(* Logix 5000 project; controller cal1615 1756-L62 rev 20.11; software revision 20.05; part 41 of 82 *)
(* tags used below, declared in another part *)
   FAULT : BOOL;   // Fault AFI
   p01_recipe_active : recipe;   // Active Recipe
   p01r02_plc_scan_time_in_sec : REAL;   // System PLC Scan Time in Seconds
   p01r09 : routine;   // System Modes
   p01r09_pb_global_reset : BOOL;   // System Modes PB: Global Fault Reset
   p01r12_master_ramped_speed : REAL;   // System Line Accel Decel Control Master Ramped Speed
   p01r13_line_running : BOOL;   // System Line Start Sequence Line Running
   p01r13_line_slow_ramp : BOOL;   // System Line Start Sequence Start Line to Slow Speed
   p01r13_permissive_drives : BOOL;   // System Line Start Sequence Permissive Drives
   p02_dint_from_hmi : hmi_dint;
   p20_acc_fill_prs : REAL;   // Upper Poly Letoff Modes A Toggle
   p20_acc_tens_prs : REAL;   // Letoff Accumulator Pressure Tension Setpoint
   p20_ai_lc01 : REAL;   // Letoff Analog Input Line Tension Load Cell Splicer
   p20_ai_loa_speed : REAL;   // Letoff Inputs Letoff A VFD Surface Speed
   p20_ao_acc_ctr_prs : REAL;   // Letoff Analog Output Accumulator Counter Pressure
   p20_ao_acc_ten_prs : REAL;   // Letoff Analog Output Accumulator Tension Pressure
   p20_ao_loa_selected_speed : REAL;   // Letoff Output Selected Speed
   p20_ao_loa_torque : REAL;
   p20_di_acc_empty : BOOL;   // Letoff Digital Input Letoff Accumulator Empty Position
   p20_di_acc_full : BOOL;   // Letoff Digital Input Letoff Accumulator Full Control Position
   p20_di_loa_active : BOOL;   // Letoff Digital Input Letoff A Active
   p20_di_loa_fwd_dir : BOOL;   // Letoff Digital Inputs PB: Letoff A Jog FWD
   p20_di_loa_jog : BOOL;   // Letoff Digital Inputs PB: Letoff A Jog REV
   p20_di_loa_start : BOOL;   // Letoff Digital Input PB: Letoff A Start
   p20_di_loa_stop : BOOL;   // Letoff Digital Input PB: Letoff A Stop Stop = 0
   p20_di_lof_acc_fill : BOOL;   // Letoff Digital Input PB: Accumulator Fill
   p20_do_acc_enable_tension : BOOL;   // Letoff Digital Output Enable Accumulator Lift Tension
   p20_do_close_nip : BOOL;   // Letoff Digital Output Feedroll Roll Nip Close
   p20_param_acc_auto_fill : REAL;
   p20_param_acc_ctr_prs : REAL;   // Letoff Parameter Carriage Counter Pressure Setpoint
   p20_param_acc_empty_prs : REAL;
   p20_param_acc_fast_accel : REAL;
   p20_param_acc_fast_decel : REAL;
   p20_param_acc_fill_ctr_prs : REAL;
   p20_param_acc_high_prs : REAL;   // Letoff Parameter High Pressure Setpoint
   p20_param_acc_init_high_prs : REAL;
   p20_param_acc_init_low_prs : REAL;
   p20_param_acc_init_prs : REAL;   // Letoff Accumulator Initial Pressure for Ramp
   p20_param_acc_med_accel : REAL;
   p20_param_acc_med_decel : REAL;
   p20_param_acc_pid_accel : REAL;
   p20_param_acc_pid_decel : REAL;
   p20_param_acc_pos_prs : REAL;
   p20_param_acc_slow_accel : REAL;
   p20_param_acc_slow_decel : REAL;
   p20_param_empty_pct : REAL;
   p20_param_high_accel_rate : REAL;
   p20_param_high_ctrl_pct : REAL;   // Letoff Parameter High Accumulator Control Position
   p20_param_high_decel_rate : REAL;
   p20_param_high_low_ctrl_pct : REAL;   // Letoff Accumulator High Control Position Low Limit
   p20_param_jog_accel_rate : REAL;
   p20_param_jog_decel_rate : REAL;
   p20_param_letoff_jog_speed : REAL;
   p20_param_lof_fast_fill : REAL;
   p20_param_lof_slow_fill : REAL;
   p20_param_lof_stop_fill : REAL;
   p20_param_low_ctrl_pct : REAL;   // Letoff Parameter Low Accumulator Control Position
   p20_param_low_low_ctrl_pct : REAL;
   p20_param_norm_accel_rate : REAL;
   p20_param_norm_decel_rate : REAL;   // Letoff Parameter Letoff A Decel Rate
   p20_param_prs_accel_rate : REAL;   // Letoff Accumulator Accel/Decel Ramp Accel Rate
   p20_param_prs_decel_rate : REAL;   // Letoff Accumulator Accel/Decel Ramp Decel Rate
   p20_param_run_torque : REAL;
   p20_vfd_di_loa : acs800_di_normal;   // Letoff A VFD Inputs
   p20_vfd_do_loa : acs800_do_normal;   // Letoff A VFD Outputs
   p20_zero_tension_prs : REAL;
   p20r01 : routine;   // Letoff Main
   p20r09_accumulator_auto : BOOL;   // Letoff Modes Accumulator Auto Mode
   p20r10_pid_psn : PID;   // Letoff Letoff Position Control PID
   p20r10_speed_offset : REAL;   // Letoff Letoff Speed Control Speed Offset
   p20r11_request_close_nip : BOOL;   // Letoff Feedroll Request Close Feedroll Nip Roll
   p20r13 : routine;   // Letoff Accum Control
   p20r13_acc_top_pos : REAL;   // Upper Poly Letoff Modes Letoff B Tension Mode
   p20r13_ai_acc_pct : REAL;   // Letoff Accumulator Pct Full
   p20r13_enc : SYS_ENC;   // Letoff Accumulator Encoder
   p20r13_ramp_tension_pressure : SYS_ACC_DEC_RAMP;   // Letoff Accumulator Tension Pressure Ramp
   p20r13_request_fill : BOOL;   // Letoff Accumulator Request Fill
   p20r13_selected_pressure : REAL;   // Letoff Accumulator Selected Pressure
   p20r13_state : DINT;   // Letoff Accumulator State
   p20r13_status : DINT;   // Letoff Accumulator Fill Status
   p20r13_timer_fault : TIMER[4];   // Letoff Accum Control Fault Delay
   p20r13_timer_warning : TIMER[4];   // Letoff Accum Control Warning Delay
   p20r14_acc_request_tension_ctrl : BOOL;   // Letoff Accumulator Fill Pressure Request Tension Control
   p20r15 : routine;   // Letoff Letoff A VFD
   p20r15_loa_accel : REAL;   // Letoff Letoff A VFD Accel Rate ORG: 100
   p20r15_loa_accel_decel_ramp : SYS_ACC_DEC_RAMP;   // Letoff Letoff A VFD Accel Decel Ramp
   p20r15_loa_decel : REAL;   // Letoff Letoff A VFD Decel Rate ORG: 20
   p20r15_loa_on : BOOL;   // Letoff Letoff A VFD On
   p20r15_loa_selected_speed : REAL;   // Letoff Letoff A VFD Selected Speed
   p20r15_permissive_run : BOOL;   // Letoff Letoff A VFD Permissive Run
   p20r15_request_jog_fwd : BOOL;   // Letoff Letoff A VFD Request Jog FWD
   p20r15_request_jog_rev : BOOL;   // Letoff Letoff A VFD Request Jog REV
   p20r15_request_over_speed : BOOL;   // Letoff Letoff A VFD Request Accumulator Over-Speed
   p20r15_request_position : BOOL;   // Letoff Letoff A VFD Request Accumulator Position Control
   p20r15_request_stop : BOOL;   // Letoff Letoff A VFD Request Stop
   p20r15_request_tension : BOOL;   // Letoff Letoff A VFD Request Tension
   p20r15_request_thread_fwd : BOOL;
   p20r15_request_thread_rev : BOOL;
   p20r15_timer_fault : TIMER[10];   // Letoff Letoff A VFD Fault Timer
   p20r15_zero_speed : BOOL;   // Letoff Letoff A VFD At Zero Speed
   p20r17_letoff_avg_diam_inch : REAL;   // Letoff Letoff Diameter Calc Average Diameter [in]
   p22_ao_selected_speed : REAL;   // Tension Stand 1 VFD Selected Speed
   p22r11_request_thread_fwd : BOOL;   // Tension Stand 1 VFD Request Thread FWD
   p22r11_request_thread_rev : BOOL;   // Tension Stand 1 VFD Request Thread REV
   p25r11_request_thread_fwd : BOOL;   // Tension Stand 2 VFD Request Thread FWD
   p25r11_request_thread_rev : BOOL;   // Tension Stand 2 VFD Request Thread REV
   p27r01 : routine;   // Winder Main
(* P20_Letoff, continued *)

ROUTINE R13_Accumulator   (* ladder *)
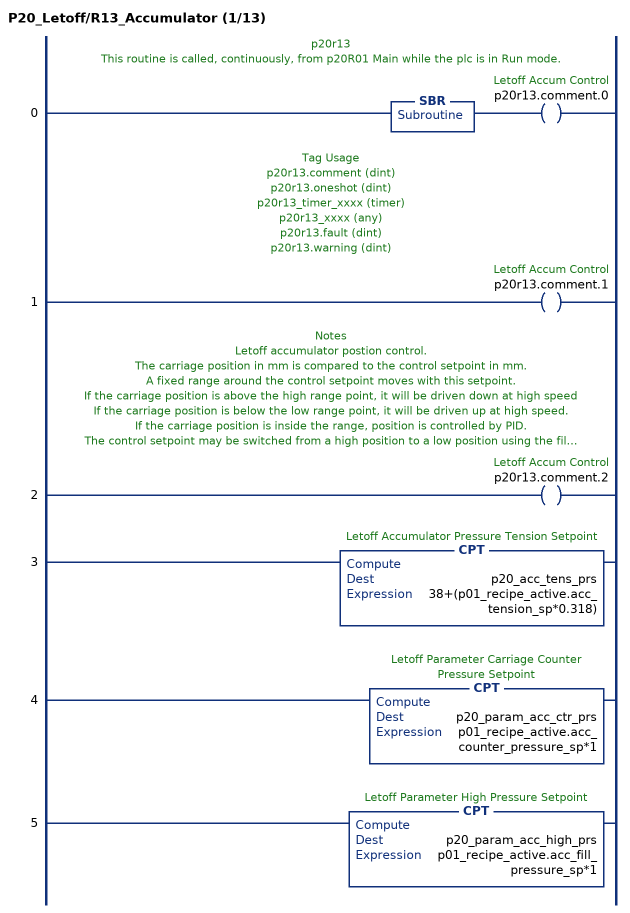
   // p20r13
   // This routine is called, continuously, from p20R01 Main while the plc is in Run mode.
   0: SBR()OTE(p20r13.comment.0);
   // Tag Usage
   // p20r13.comment (dint)
   // p20r13.oneshot (dint)
   // p20r13_timer_xxxx (timer)
   // p20r13_xxxx (any)
   // p20r13.fault (dint)
   // p20r13.warning (dint)
   1: OTE(p20r13.comment.1);
   // Notes
   // Letoff accumulator postion control.
   // The carriage position in mm is compared to the control setpoint in mm.
   // A fixed range around the control setpoint moves with this setpoint.
   // If the carriage position is above the high range point, it will be driven down at high speed
   // If the carriage position is below the low range point, it will be driven up at high speed.
   // If the carriage position is inside the range, position is controlled by PID.
   // The control setpoint may be switched from a high position to a low position using the fill accumulator function.
   2: OTE(p20r13.comment.2);
   3: CPT(p20_acc_tens_prs,38+(p01_recipe_active.acc_tension_sp*0.318));
   4: CPT(p20_param_acc_ctr_prs,p01_recipe_active.acc_counter_pressure_sp*1);
   5: CPT(p20_param_acc_high_prs,p01_recipe_active.acc_fill_pressure_sp*1);
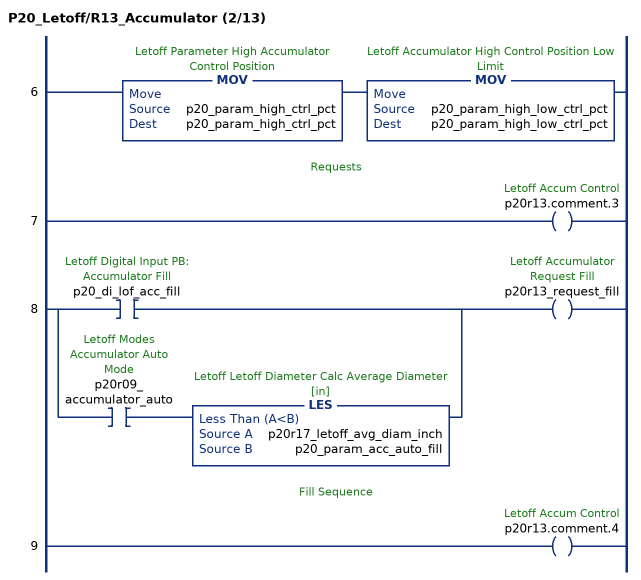
   6: MOV(p20_param_high_ctrl_pct,p20_param_high_ctrl_pct)MOV(p20_param_high_low_ctrl_pct,p20_param_high_low_ctrl_pct);
   // Requests
   7: OTE(p20r13.comment.3);
   8: [XIC(p20_di_lof_acc_fill) ,XIC(p20r09_accumulator_auto) LES(p20r17_letoff_avg_diam_inch,p20_param_acc_auto_fill) ]OTE(p20r13_request_fill);
   // Fill Sequence
   9: OTE(p20r13.comment.4);
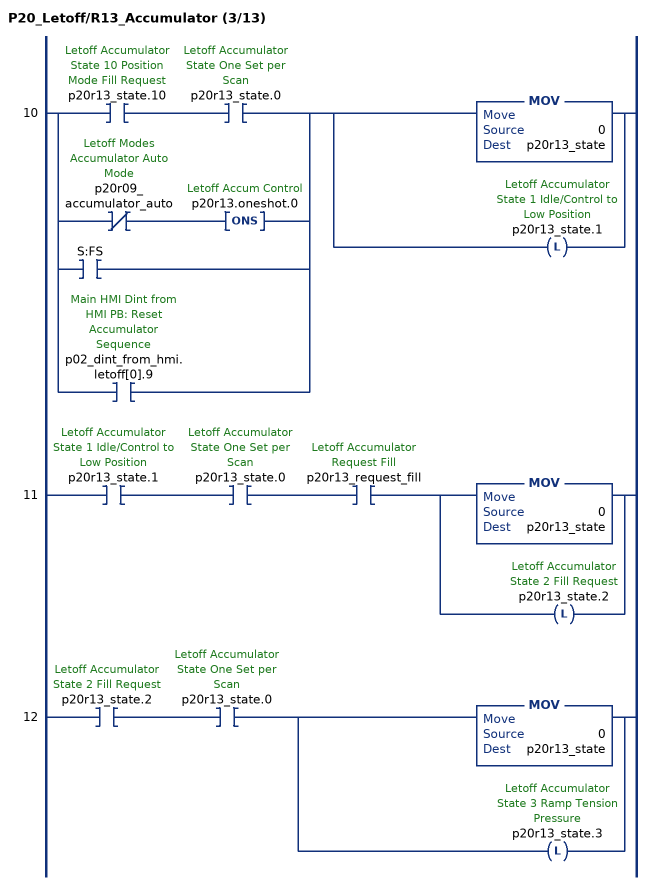
   10: [XIC(p20r13_state.10) XIC(p20r13_state.0) ,XIO(p20r09_accumulator_auto) ONS(p20r13.oneshot.0) ,XIC(S:FS) ,XIC(p02_dint_from_hmi.letoff[0].9) ][MOV(0,p20r13_state) ,OTL(p20r13_state.1) ];
   11: XIC(p20r13_state.1)XIC(p20r13_state.0)XIC(p20r13_request_fill)[MOV(0,p20r13_state) ,OTL(p20r13_state.2) ];
   12: XIC(p20r13_state.2)XIC(p20r13_state.0)[MOV(0,p20r13_state) ,OTL(p20r13_state.3) ];
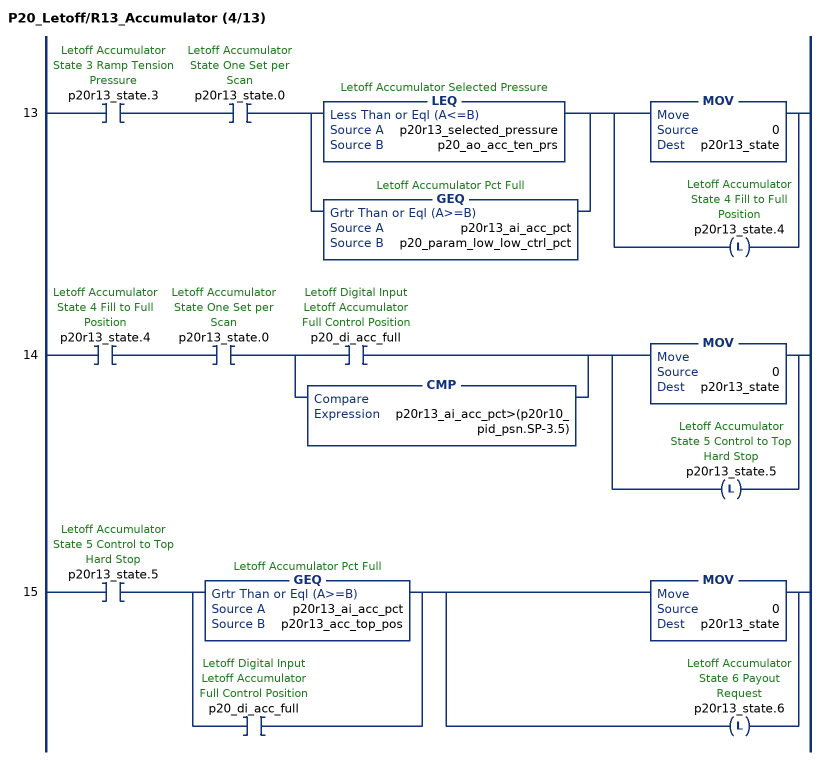
   13: XIC(p20r13_state.3)XIC(p20r13_state.0)[LEQ(p20r13_selected_pressure,p20_ao_acc_ten_prs) ,GEQ(p20r13_ai_acc_pct,p20_param_low_low_ctrl_pct) ][MOV(0,p20r13_state) ,OTL(p20r13_state.4) ];
   14: XIC(p20r13_state.4)XIC(p20r13_state.0)[XIC(p20_di_acc_full) ,CMP(p20r13_ai_acc_pct>(p20r10_pid_psn.SP-3.5)) ][MOV(0,p20r13_state) ,OTL(p20r13_state.5) ];
   15: XIC(p20r13_state.5)[GEQ(p20r13_ai_acc_pct,p20r13_acc_top_pos) ,XIC(p20_di_acc_full) ][MOV(0,p20r13_state) ,OTL(p20r13_state.6) ];
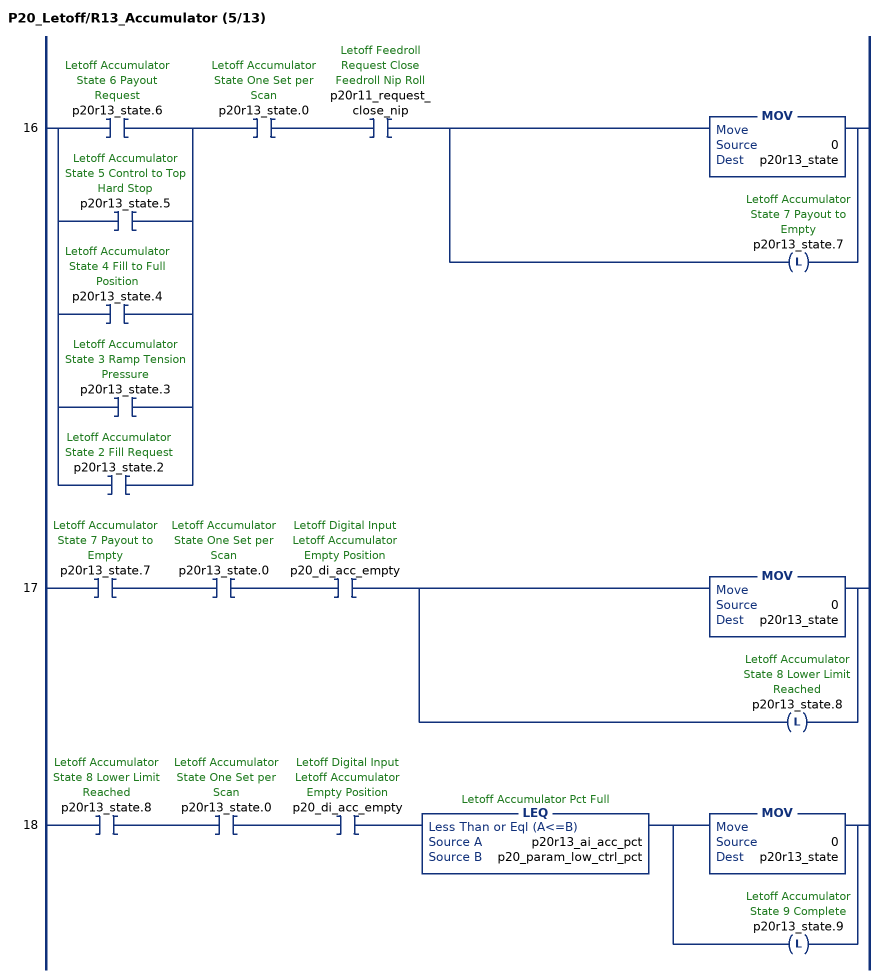
   16: [XIC(p20r13_state.6) ,XIC(p20r13_state.5) ,XIC(p20r13_state.4) ,XIC(p20r13_state.3) ,XIC(p20r13_state.2) ]XIC(p20r13_state.0)XIC(p20r11_request_close_nip)[MOV(0,p20r13_state) ,OTL(p20r13_state.7) ];
   17: XIC(p20r13_state.7)XIC(p20r13_state.0)XIC(p20_di_acc_empty)[MOV(0,p20r13_state) ,OTL(p20r13_state.8) ];
   18: XIC(p20r13_state.8)XIC(p20r13_state.0)XIC(p20_di_acc_empty)LEQ(p20r13_ai_acc_pct,p20_param_low_ctrl_pct)[MOV(0,p20r13_state) ,OTL(p20r13_state.9) ];
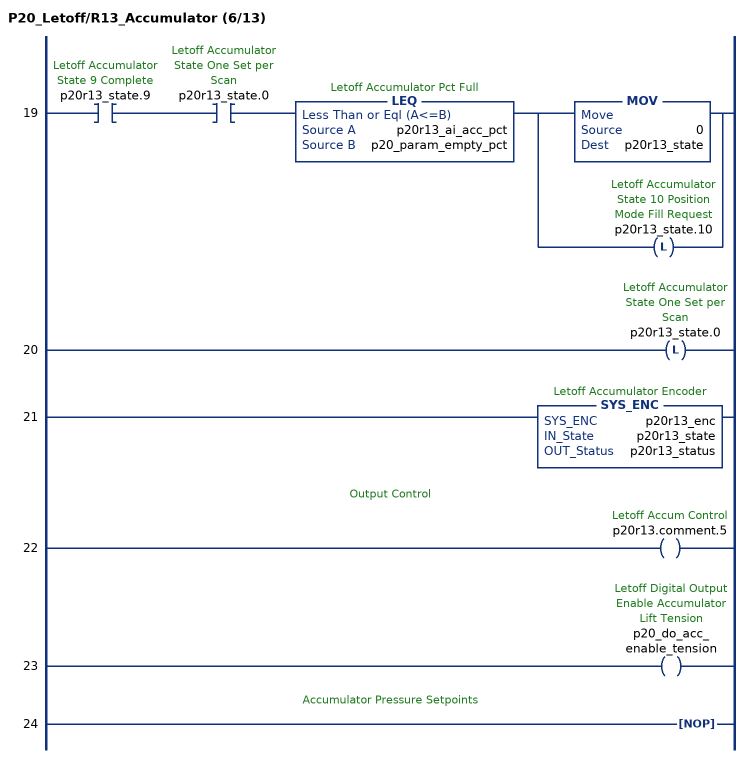
   19: XIC(p20r13_state.9)XIC(p20r13_state.0)LEQ(p20r13_ai_acc_pct,p20_param_empty_pct)[MOV(0,p20r13_state) ,OTL(p20r13_state.10) ];
   20: OTL(p20r13_state.0);
   21: SYS_ENC(p20r13_enc,p20r13_state,p20r13_status);
   // Output Control
   22: OTE(p20r13.comment.5);
   23: OTE(p20_do_acc_enable_tension);
   // Accumulator Pressure Setpoints
   24: NOP();
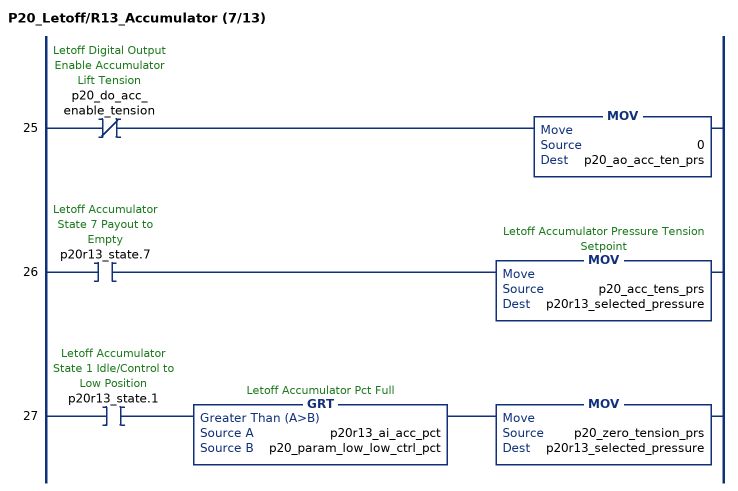
   25: XIO(p20_do_acc_enable_tension)MOV(0,p20_ao_acc_ten_prs);
   26: XIC(p20r13_state.7)MOV(p20_acc_tens_prs,p20r13_selected_pressure);
   27: XIC(p20r13_state.1)GRT(p20r13_ai_acc_pct,p20_param_low_low_ctrl_pct)MOV(p20_zero_tension_prs,p20r13_selected_pressure);
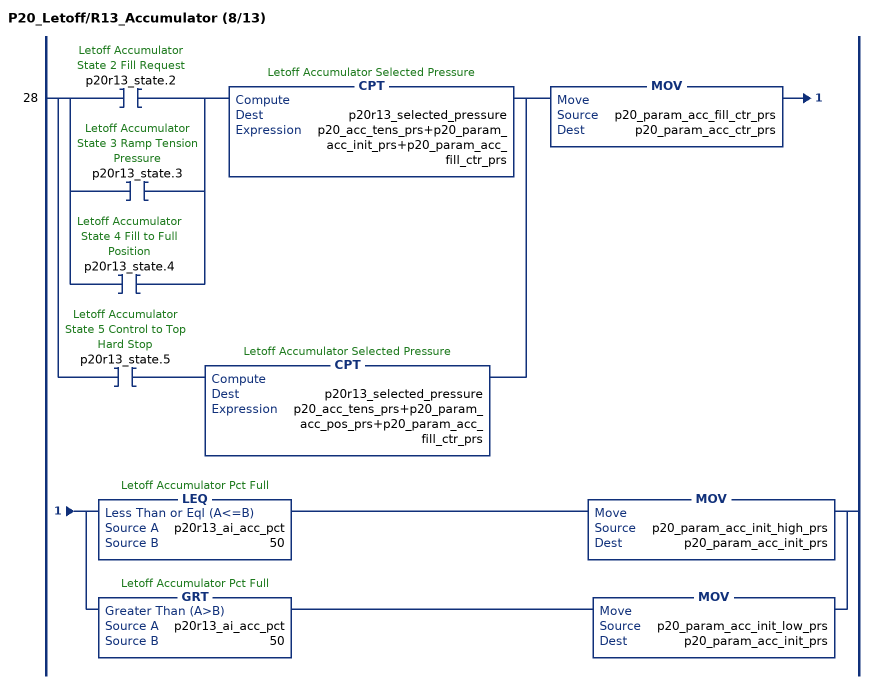
   28: [[XIC(p20r13_state.2) ,XIC(p20r13_state.3) ,XIC(p20r13_state.4) ] CPT(p20r13_selected_pressure,p20_acc_tens_prs+p20_param_acc_init_prs+p20_param_acc_fill_ctr_prs) ,XIC(p20r13_state.5) CPT(p20r13_selected_pressure,p20_acc_tens_prs+p20_param_acc_pos_prs+p20_param_acc_fill_ctr_prs) ]MOV(p20_param_acc_fill_ctr_prs,p20_param_acc_ctr_prs)[LEQ(p20r13_ai_acc_pct,50) MOV(p20_param_acc_init_high_prs,p20_param_acc_init_prs) ,GRT(p20r13_ai_acc_pct,50) MOV(p20_param_acc_init_low_prs,p20_param_acc_init_prs) ];
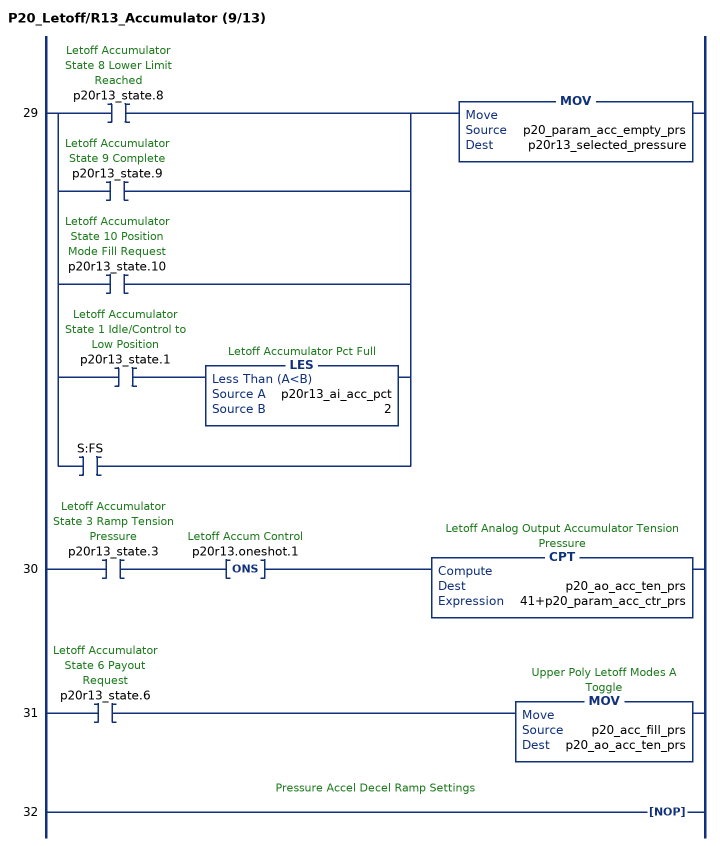
   29: [XIC(p20r13_state.8) ,XIC(p20r13_state.9) ,XIC(p20r13_state.10) ,XIC(p20r13_state.1) LES(p20r13_ai_acc_pct,2) ,XIC(S:FS) ]MOV(p20_param_acc_empty_prs,p20r13_selected_pressure);
   30: XIC(p20r13_state.3)ONS(p20r13.oneshot.1)CPT(p20_ao_acc_ten_prs,41+p20_param_acc_ctr_prs);
   31: XIC(p20r13_state.6)MOV(p20_acc_fill_prs,p20_ao_acc_ten_prs);
   // Pressure Accel Decel Ramp Settings
   32: NOP();
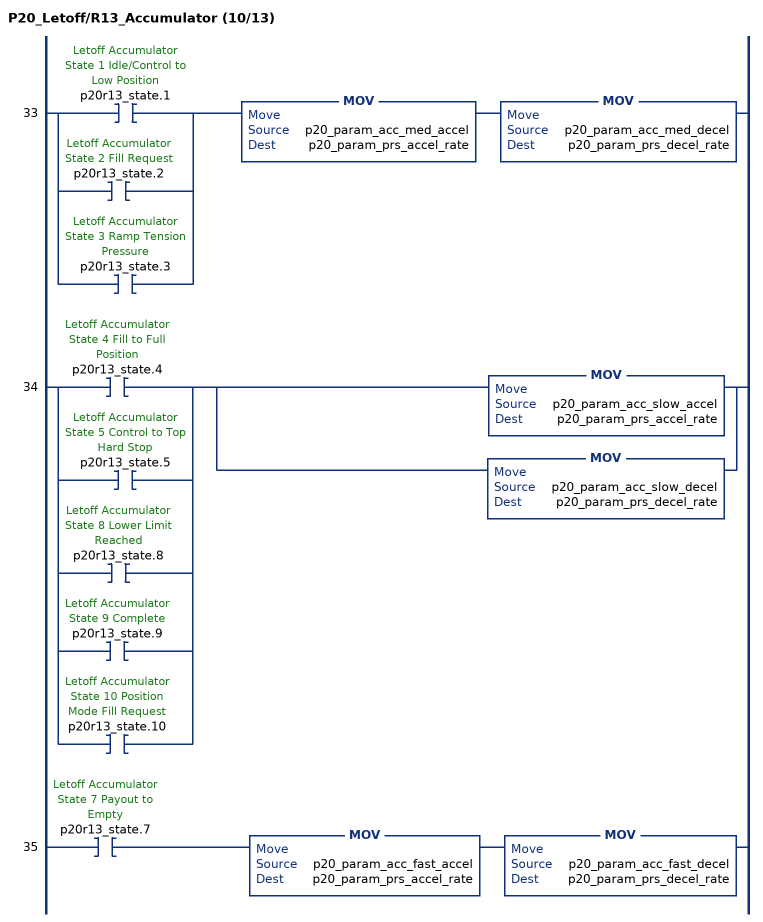
   33: [XIC(p20r13_state.1) ,XIC(p20r13_state.2) ,XIC(p20r13_state.3) ]MOV(p20_param_acc_med_accel,p20_param_prs_accel_rate)MOV(p20_param_acc_med_decel,p20_param_prs_decel_rate);
   34: [XIC(p20r13_state.4) ,XIC(p20r13_state.5) ,XIC(p20r13_state.8) ,XIC(p20r13_state.9) ,XIC(p20r13_state.10) ][MOV(p20_param_acc_slow_accel,p20_param_prs_accel_rate) ,MOV(p20_param_acc_slow_decel,p20_param_prs_decel_rate) ];
   35: XIC(p20r13_state.7)MOV(p20_param_acc_fast_accel,p20_param_prs_accel_rate)MOV(p20_param_acc_fast_decel,p20_param_prs_decel_rate);
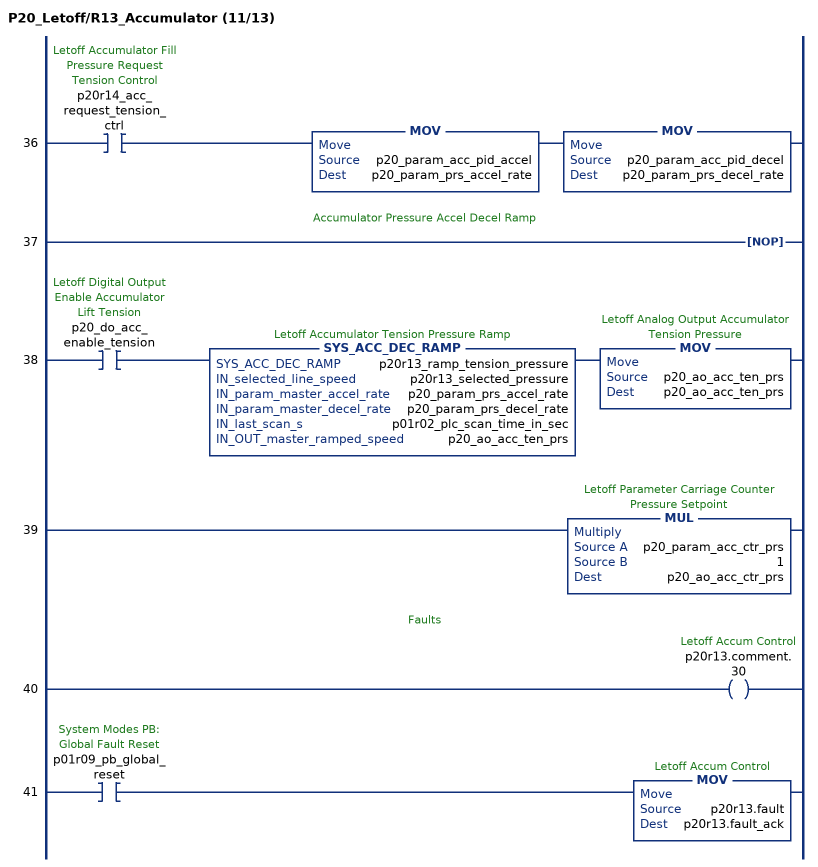
   36: XIC(p20r14_acc_request_tension_ctrl)MOV(p20_param_acc_pid_accel,p20_param_prs_accel_rate)MOV(p20_param_acc_pid_decel,p20_param_prs_decel_rate);
   // Accumulator Pressure Accel Decel Ramp
   37: NOP();
   38: XIC(p20_do_acc_enable_tension)SYS_ACC_DEC_RAMP(p20r13_ramp_tension_pressure,p20r13_selected_pressure,p20_param_prs_accel_rate,p20_param_prs_decel_rate,p01r02_plc_scan_time_in_sec,p20_ao_acc_ten_prs)MOV(p20_ao_acc_ten_prs,p20_ao_acc_ten_prs);
   39: MUL(p20_param_acc_ctr_prs,1,p20_ao_acc_ctr_prs);
   // Faults
   40: OTE(p20r13.comment.30);
   41: XIC(p01r09_pb_global_reset)MOV(p20r13.fault,p20r13.fault_ack);
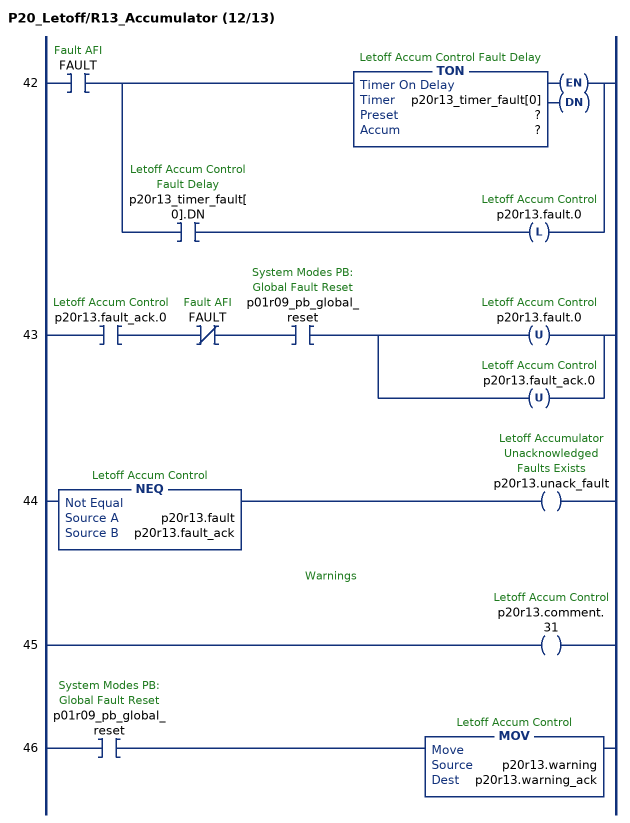
   42: XIC(FAULT)[TON(p20r13_timer_fault[0],?,?) ,XIC(p20r13_timer_fault[0].DN) OTL(p20r13.fault.0) ];
   43: XIC(p20r13.fault_ack.0)XIO(FAULT)XIC(p01r09_pb_global_reset)[OTU(p20r13.fault.0) ,OTU(p20r13.fault_ack.0) ];
   44: NEQ(p20r13.fault,p20r13.fault_ack)OTE(p20r13.unack_fault);
   // Warnings
   45: OTE(p20r13.comment.31);
   46: XIC(p01r09_pb_global_reset)MOV(p20r13.warning,p20r13.warning_ack);
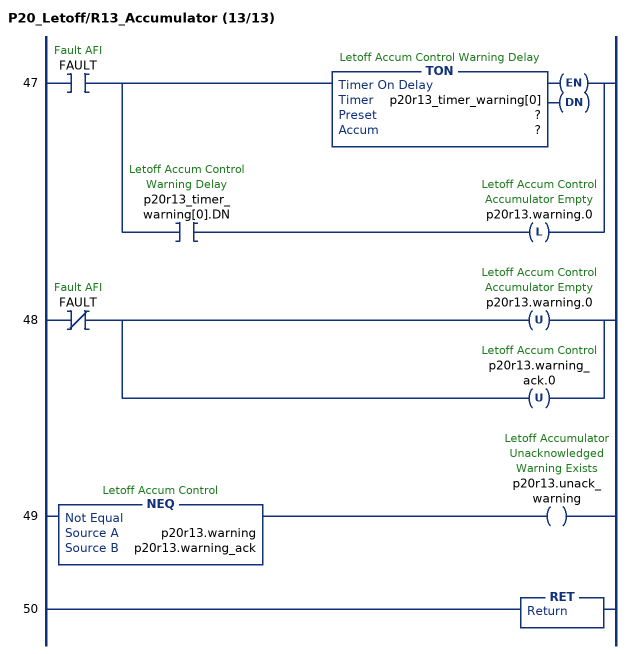
   47: XIC(FAULT)[TON(p20r13_timer_warning[0],?,?) ,XIC(p20r13_timer_warning[0].DN) OTL(p20r13.warning.0) ];
   48: XIO(FAULT)[OTU(p20r13.warning.0) ,OTU(p20r13.warning_ack.0) ];
   49: NEQ(p20r13.warning,p20r13.warning_ack)OTE(p20r13.unack_warning);
   50: RET();
END_ROUTINE

ROUTINE R15_Letoff_A_VFD   (* ladder *)
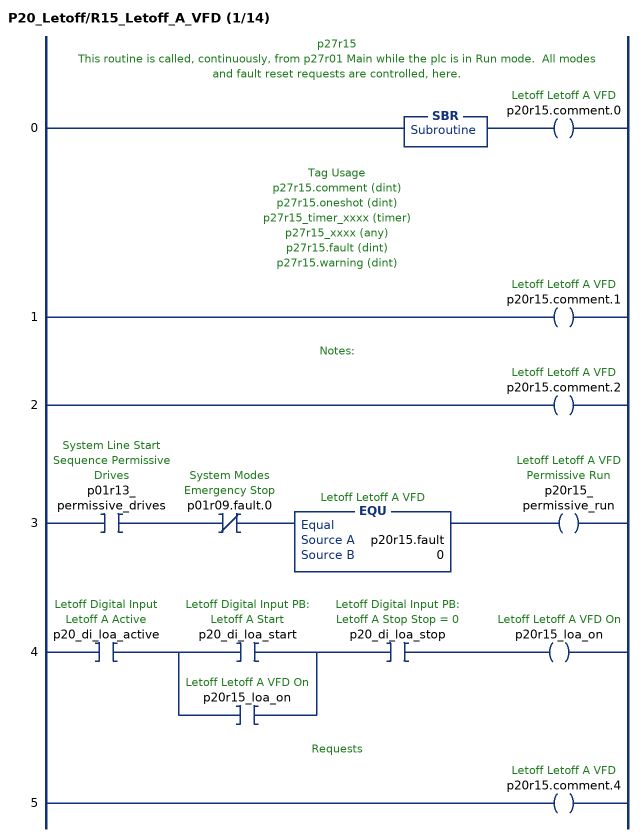
   // p27r15
   // This routine is called, continuously, from p27r01 Main while the plc is in Run mode.  All modes and fault reset requests are controlled, here.
   0: SBR()OTE(p20r15.comment.0);
   // Tag Usage
   // p27r15.comment (dint)
   // p27r15.oneshot (dint)
   // p27r15_timer_xxxx (timer)
   // p27r15_xxxx (any)
   // p27r15.fault (dint)
   // p27r15.warning (dint)
   1: OTE(p20r15.comment.1);
   // Notes:
   2: OTE(p20r15.comment.2);
   3: XIC(p01r13_permissive_drives)XIO(p01r09.fault.0)EQU(p20r15.fault,0)OTE(p20r15_permissive_run);
   4: XIC(p20_di_loa_active)[XIC(p20_di_loa_start) ,XIC(p20r15_loa_on) ]XIC(p20_di_loa_stop)OTE(p20r15_loa_on);
   // Requests
   5: OTE(p20r15.comment.4);
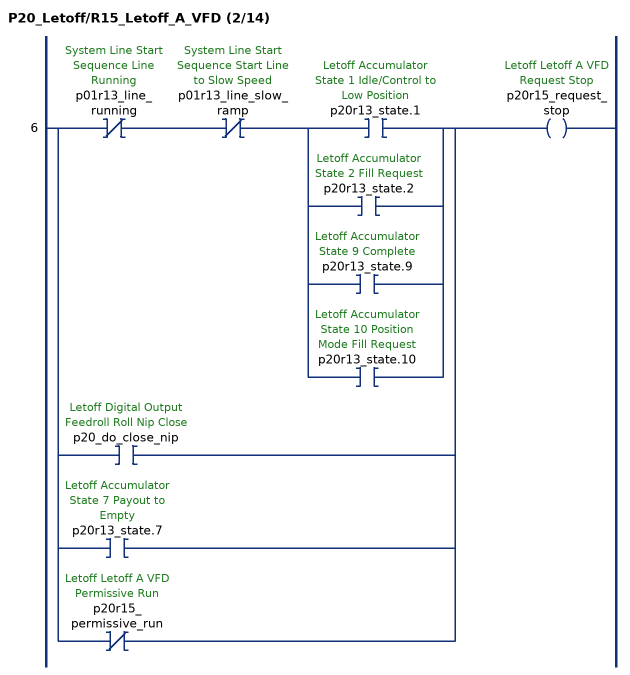
   6: [XIO(p01r13_line_running) XIO(p01r13_line_slow_ramp) [XIC(p20r13_state.1) ,XIC(p20r13_state.2) ,XIC(p20r13_state.9) ,XIC(p20r13_state.10) ] ,XIC(p20_do_close_nip) ,XIC(p20r13_state.7) ,XIO(p20r15_permissive_run) ]OTE(p20r15_request_stop);
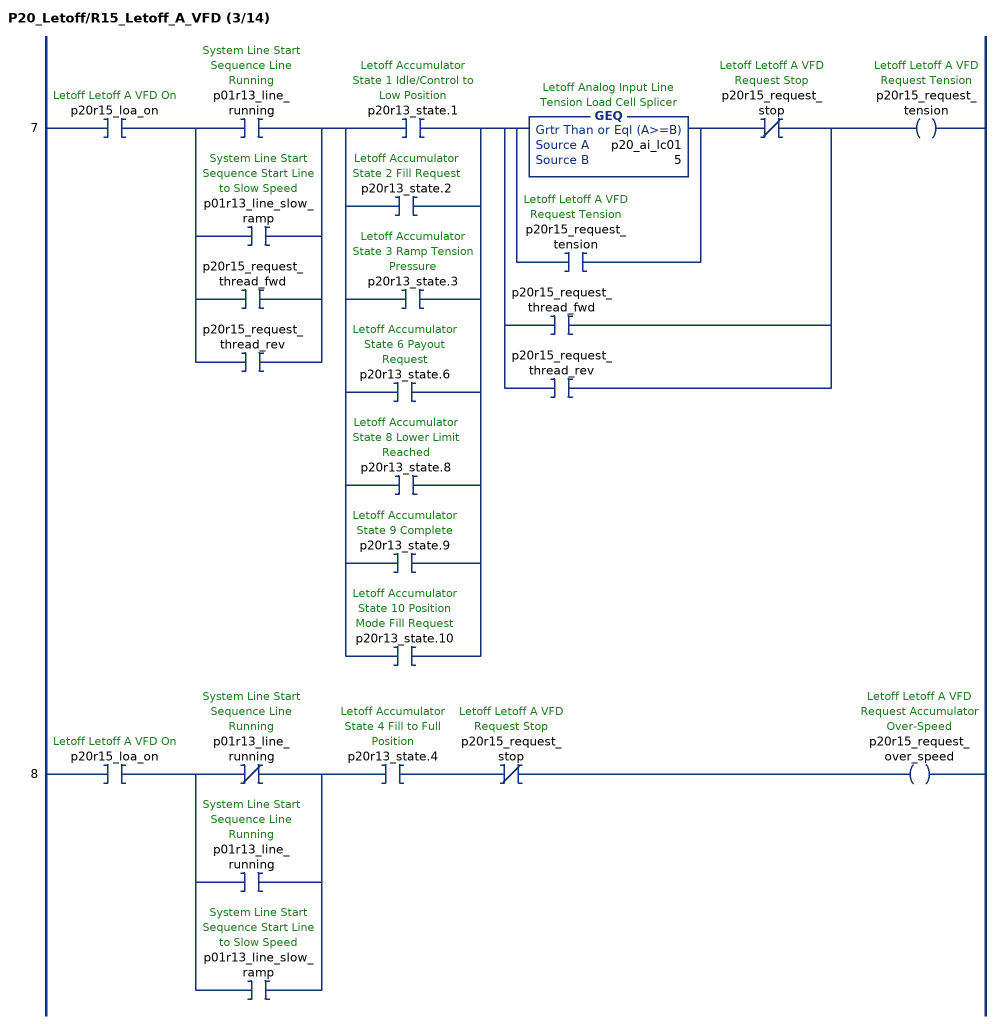
   7: XIC(p20r15_loa_on)[XIC(p01r13_line_running) ,XIC(p01r13_line_slow_ramp) ,XIC(p20r15_request_thread_fwd) ,XIC(p20r15_request_thread_rev) ][XIC(p20r13_state.1) ,XIC(p20r13_state.2) ,XIC(p20r13_state.3) ,XIC(p20r13_state.6) ,XIC(p20r13_state.8) ,XIC(p20r13_state.9) ,XIC(p20r13_state.10) ][[GEQ(p20_ai_lc01,5) ,XIC(p20r15_request_tension) ] XIO(p20r15_request_stop) ,XIC(p20r15_request_thread_fwd) ,XIC(p20r15_request_thread_rev) ]OTE(p20r15_request_tension);
   8: XIC(p20r15_loa_on)[XIO(p01r13_line_running) ,XIC(p01r13_line_running) ,XIC(p01r13_line_slow_ramp) ]XIC(p20r13_state.4)XIO(p20r15_request_stop)OTE(p20r15_request_over_speed);
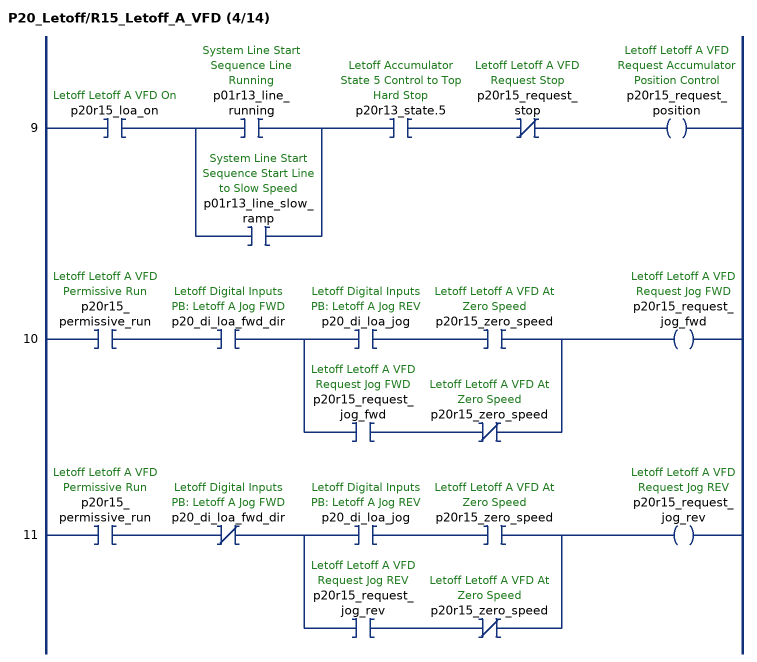
   9: XIC(p20r15_loa_on)[XIC(p01r13_line_running) ,XIC(p01r13_line_slow_ramp) ]XIC(p20r13_state.5)XIO(p20r15_request_stop)OTE(p20r15_request_position);
   10: XIC(p20r15_permissive_run)XIC(p20_di_loa_fwd_dir)[XIC(p20_di_loa_jog) XIC(p20r15_zero_speed) ,XIC(p20r15_request_jog_fwd) XIO(p20r15_zero_speed) ]OTE(p20r15_request_jog_fwd);
   11: XIC(p20r15_permissive_run)XIO(p20_di_loa_fwd_dir)[XIC(p20_di_loa_jog) XIC(p20r15_zero_speed) ,XIC(p20r15_request_jog_rev) XIO(p20r15_zero_speed) ]OTE(p20r15_request_jog_rev);
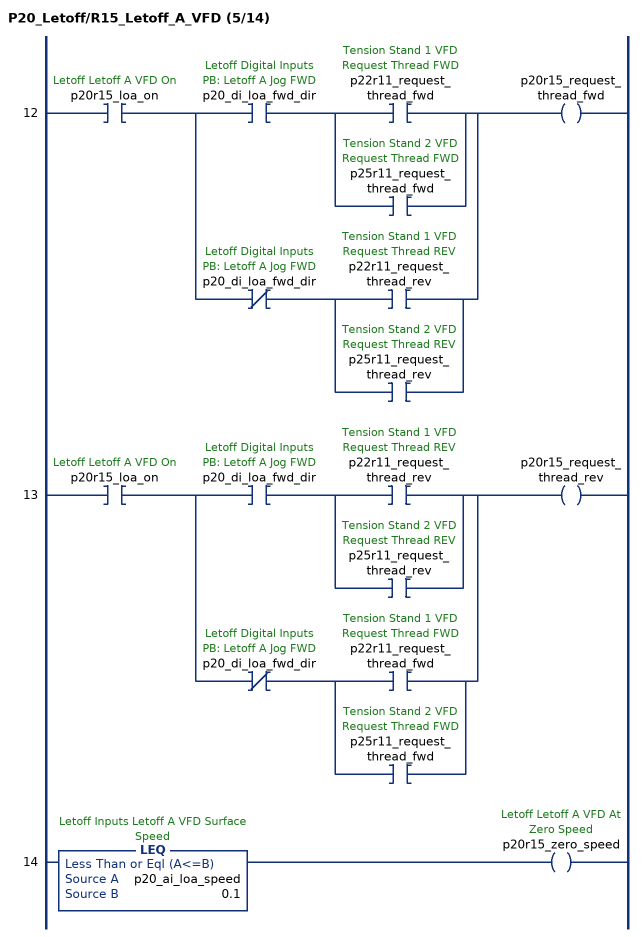
   12: XIC(p20r15_loa_on)[XIC(p20_di_loa_fwd_dir) [XIC(p22r11_request_thread_fwd) ,XIC(p25r11_request_thread_fwd) ] ,XIO(p20_di_loa_fwd_dir) [XIC(p22r11_request_thread_rev) ,XIC(p25r11_request_thread_rev) ] ]OTE(p20r15_request_thread_fwd);
   13: XIC(p20r15_loa_on)[XIC(p20_di_loa_fwd_dir) [XIC(p22r11_request_thread_rev) ,XIC(p25r11_request_thread_rev) ] ,XIO(p20_di_loa_fwd_dir) [XIC(p22r11_request_thread_fwd) ,XIC(p25r11_request_thread_fwd) ] ]OTE(p20r15_request_thread_rev);
   14: LEQ(p20_ai_loa_speed,0.1)OTE(p20r15_zero_speed);
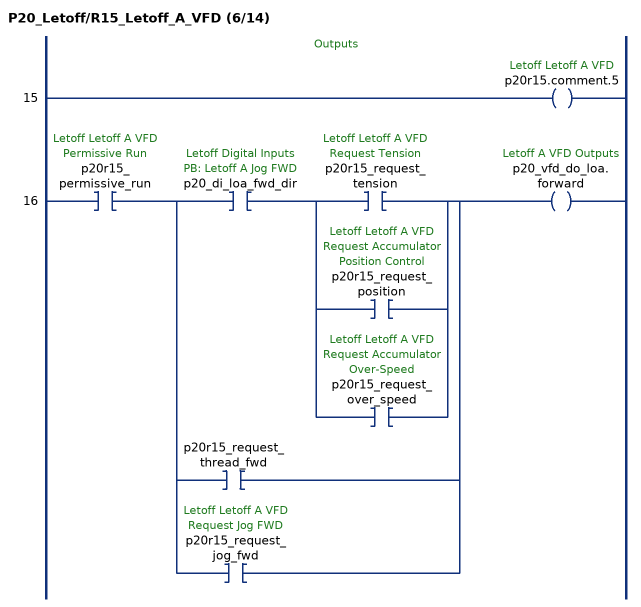
   // Outputs
   15: OTE(p20r15.comment.5);
   16: XIC(p20r15_permissive_run)[XIC(p20_di_loa_fwd_dir) [XIC(p20r15_request_tension) ,XIC(p20r15_request_position) ,XIC(p20r15_request_over_speed) ] ,XIC(p20r15_request_thread_fwd) ,XIC(p20r15_request_jog_fwd) ]OTE(p20_vfd_do_loa.forward);
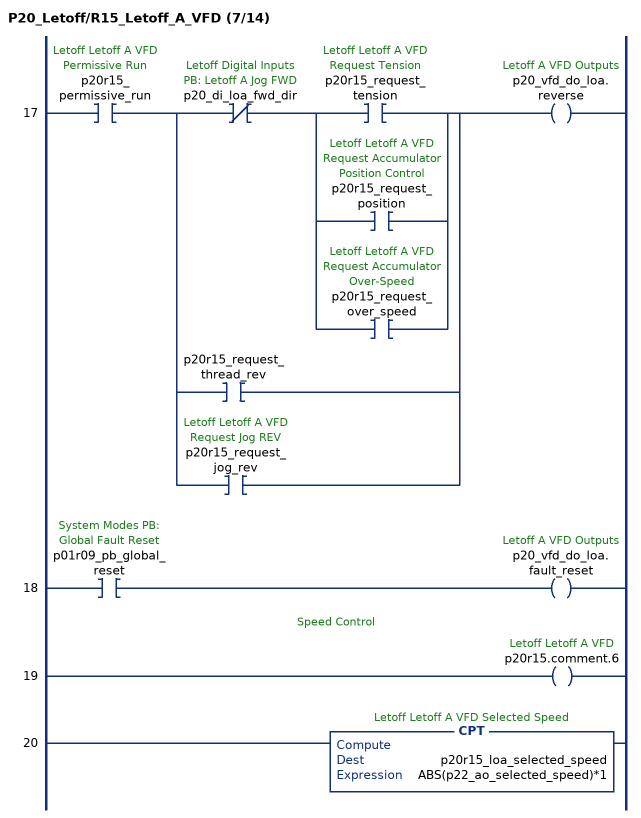
   17: XIC(p20r15_permissive_run)[XIO(p20_di_loa_fwd_dir) [XIC(p20r15_request_tension) ,XIC(p20r15_request_position) ,XIC(p20r15_request_over_speed) ] ,XIC(p20r15_request_thread_rev) ,XIC(p20r15_request_jog_rev) ]OTE(p20_vfd_do_loa.reverse);
   18: XIC(p01r09_pb_global_reset)OTE(p20_vfd_do_loa.fault_reset);
   // Speed Control
   19: OTE(p20r15.comment.6);
   20: CPT(p20r15_loa_selected_speed,ABS(p22_ao_selected_speed)*1);
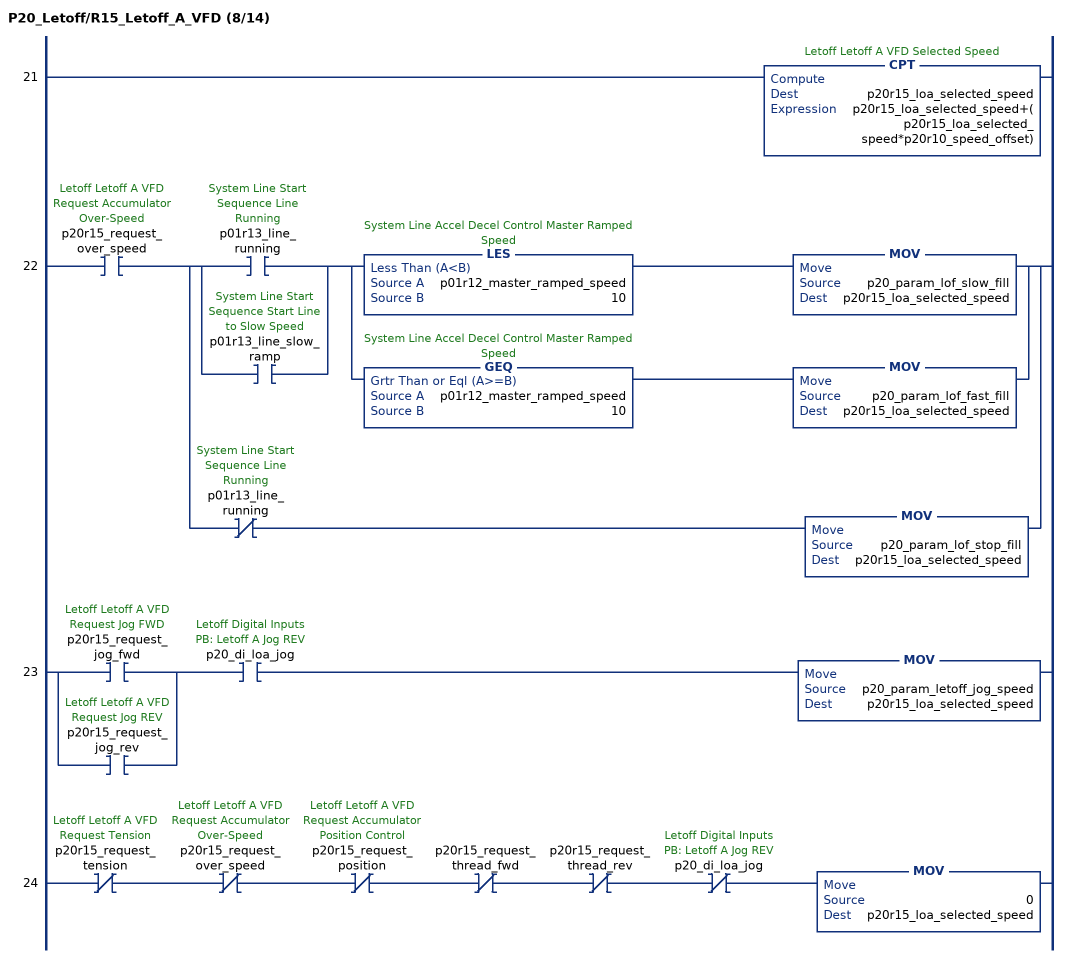
   21: CPT(p20r15_loa_selected_speed,p20r15_loa_selected_speed+(p20r15_loa_selected_speed*p20r10_speed_offset));
   22: XIC(p20r15_request_over_speed)[[XIC(p01r13_line_running) ,XIC(p01r13_line_slow_ramp) ] [LES(p01r12_master_ramped_speed,10) MOV(p20_param_lof_slow_fill,p20r15_loa_selected_speed) ,GEQ(p01r12_master_ramped_speed,10) MOV(p20_param_lof_fast_fill,p20r15_loa_selected_speed) ] ,XIO(p01r13_line_running) MOV(p20_param_lof_stop_fill,p20r15_loa_selected_speed) ];
   23: [XIC(p20r15_request_jog_fwd) ,XIC(p20r15_request_jog_rev) ]XIC(p20_di_loa_jog)MOV(p20_param_letoff_jog_speed,p20r15_loa_selected_speed);
   24: XIO(p20r15_request_tension)XIO(p20r15_request_over_speed)XIO(p20r15_request_position)XIO(p20r15_request_thread_fwd)XIO(p20r15_request_thread_rev)XIO(p20_di_loa_jog)MOV(0,p20r15_loa_selected_speed);
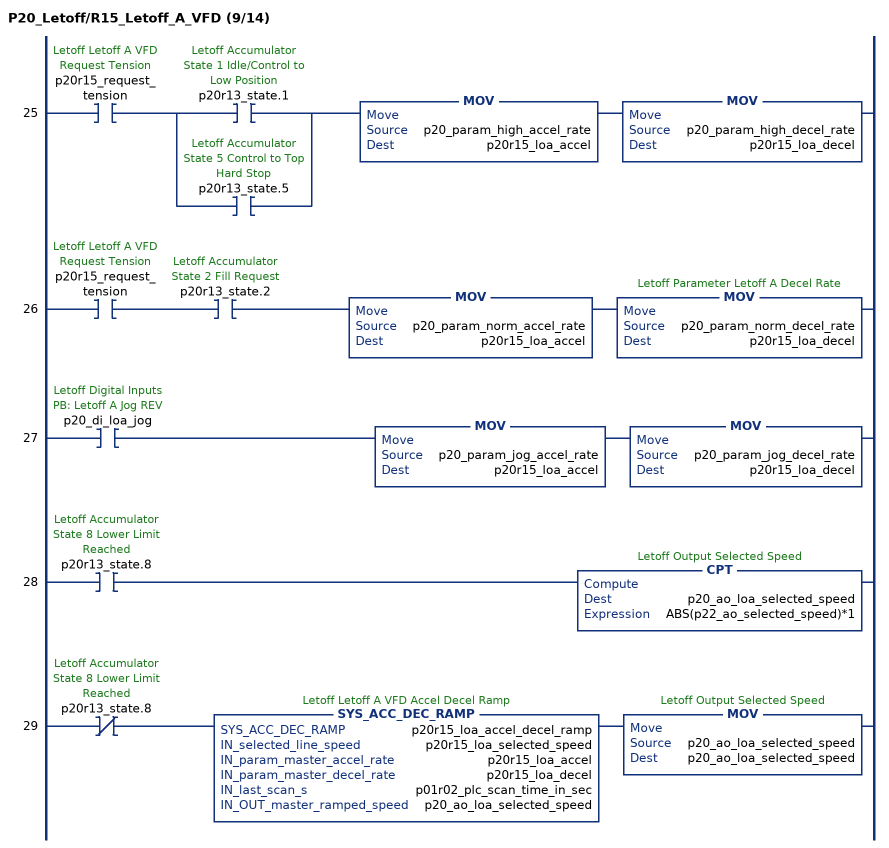
   25: XIC(p20r15_request_tension)[XIC(p20r13_state.1) ,XIC(p20r13_state.5) ]MOV(p20_param_high_accel_rate,p20r15_loa_accel)MOV(p20_param_high_decel_rate,p20r15_loa_decel);
   26: XIC(p20r15_request_tension)XIC(p20r13_state.2)MOV(p20_param_norm_accel_rate,p20r15_loa_accel)MOV(p20_param_norm_decel_rate,p20r15_loa_decel);
   27: XIC(p20_di_loa_jog)MOV(p20_param_jog_accel_rate,p20r15_loa_accel)MOV(p20_param_jog_decel_rate,p20r15_loa_decel);
   28: XIC(p20r13_state.8)CPT(p20_ao_loa_selected_speed,ABS(p22_ao_selected_speed)*1);
   29: XIO(p20r13_state.8)SYS_ACC_DEC_RAMP(p20r15_loa_accel_decel_ramp,p20r15_loa_selected_speed,p20r15_loa_accel,p20r15_loa_decel,p01r02_plc_scan_time_in_sec,p20_ao_loa_selected_speed)MOV(p20_ao_loa_selected_speed,p20_ao_loa_selected_speed);
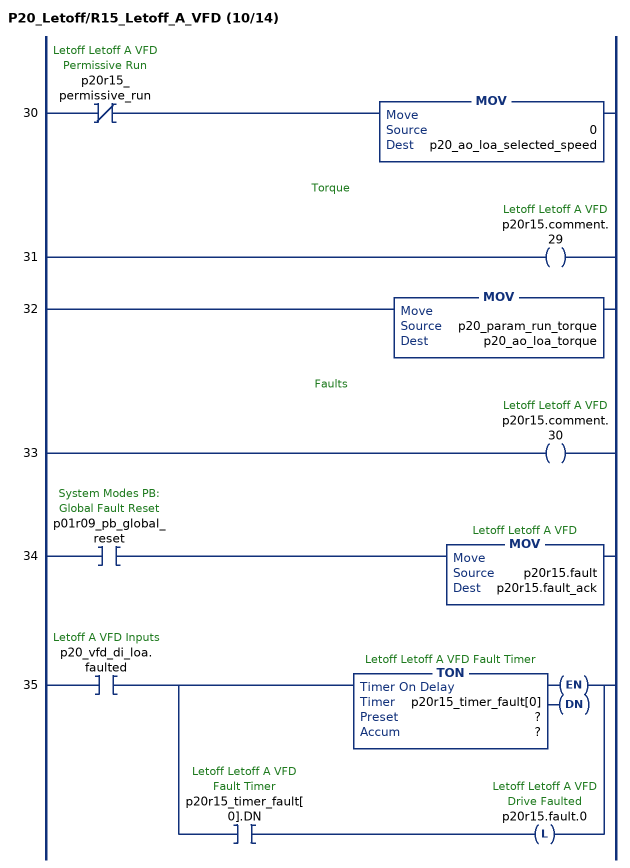
   30: XIO(p20r15_permissive_run)MOV(0,p20_ao_loa_selected_speed);
   // Torque
   31: OTE(p20r15.comment.29);
   32: MOV(p20_param_run_torque,p20_ao_loa_torque);
   // Faults
   33: OTE(p20r15.comment.30);
   34: XIC(p01r09_pb_global_reset)MOV(p20r15.fault,p20r15.fault_ack);
   35: XIC(p20_vfd_di_loa.faulted)[TON(p20r15_timer_fault[0],?,?) ,XIC(p20r15_timer_fault[0].DN) OTL(p20r15.fault.0) ];
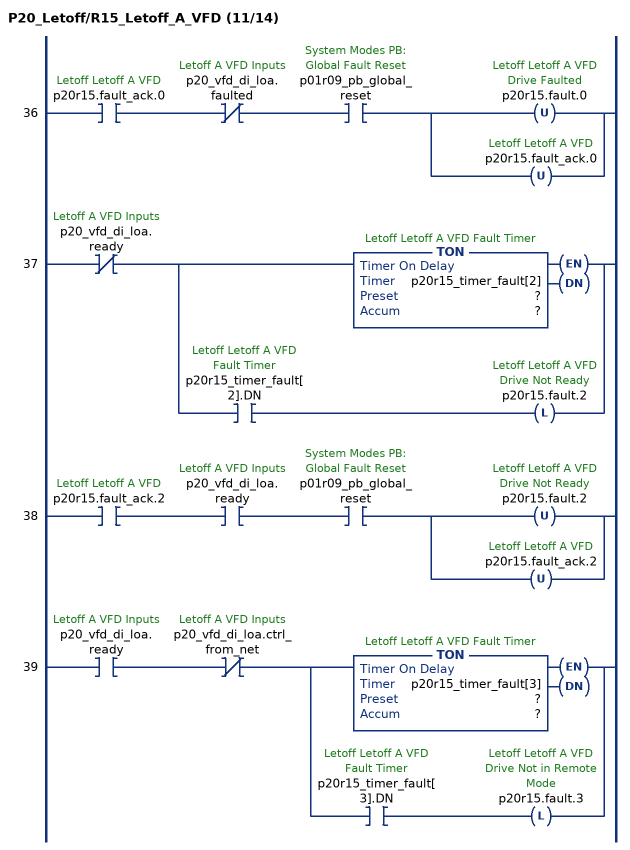
   36: XIC(p20r15.fault_ack.0)XIO(p20_vfd_di_loa.faulted)XIC(p01r09_pb_global_reset)[OTU(p20r15.fault.0) ,OTU(p20r15.fault_ack.0) ];
   37: XIO(p20_vfd_di_loa.ready)[TON(p20r15_timer_fault[2],?,?) ,XIC(p20r15_timer_fault[2].DN) OTL(p20r15.fault.2) ];
   38: XIC(p20r15.fault_ack.2)XIC(p20_vfd_di_loa.ready)XIC(p01r09_pb_global_reset)[OTU(p20r15.fault.2) ,OTU(p20r15.fault_ack.2) ];
   39: XIC(p20_vfd_di_loa.ready)XIO(p20_vfd_di_loa.ctrl_from_net)[TON(p20r15_timer_fault[3],?,?) ,XIC(p20r15_timer_fault[3].DN) OTL(p20r15.fault.3) ];
